FUNCTION_BLOCK RemoveAllMoverFromGroup EXTENDS TaskBase
VAR_INPUT
END_VAR
VAR_OUTPUT
END_VAR
VAR
	RemoveAllFromGrp			: MC_UngroupAllAxes;
	_caGroup			: ICollisionGroup;
	_removeAllMovers : BOOL;
	_errorId: UDINT;
	Logger : TcMessage_Ext;
END_VAR

METHOD Abort : BOOL
RemoveAllFromGrp.Execute := FALSE;
Abort := true;
State := 0;
END_METHOD

METHOD Cycle : BOOL
VAR_INPUT
END_VAR
CASE State OF
	0:
		IF _removeAllMovers THEN
			_done := FALSE;
			_error := FALSE;
			_busy := TRUE;
			RemoveAllFromGrp.Execute := TRUE;
			IF RemoveAllFromGrp.Busy THEN
				_removeAllMovers := FALSE;
				State := 10;
				logger.Send(TC_EVENTS.XtsCAGroupEvents.CAGroupRemoving,'');
			END_IF
		END_IF
		
	10:
		IF NOT RemoveAllFromGrp.Busy THEN
			IF RemoveAllFromGrp.Done THEN
				_done := TRUE;
				logger.Send(TC_EVENTS.XtsCAGroupEvents.AllMoversRemoved,'');
			ELSIF RemoveAllFromGrp.Error THEN
				_error := TRUE;
				_errorId := RemoveAllFromGrp.ErrorId;
				Logger.Send(TC_EVENTS.XtsCAGroupEvents.CAGroupRemoveError,'');
			END_IF
			_busy := FALSE;
			RemoveAllFromGrp.Execute := false;
			State := 0;
		END_IF
END_CASE


RemoveAllFromGrp(AxesGroup := _caGroup.GroupRef);
END_METHOD

METHOD FB_init : BOOL
VAR_INPUT
	bInitRetains : BOOL; // if TRUE, the retain variables are initialized (warm start / cold start)
	bInCopyCode : BOOL;  // if TRUE, the instance afterwards gets moved into the copy code (online change)
	CAGroup : ICollisionGroup;	
END_VAR
_caGroup := CAGroup;
END_METHOD

METHOD RemoveAllMover : BOOL
RemoveAllMover := _removeAllMovers := true;
END_METHOD

END_FUNCTION_BLOCK

(* stored: Version 1.1.0.1, ProductVersion 3.1.4024.12
   POU RemoveAllMoverFromGroup: Id {1511d483-7397-4cd0-a6db-08dd652e8cbb}, SpecialFunc None
   Method Abort: Id {e7050a73-9e5f-49ae-8033-79483a14dcd8}
   Method Cycle: Id {c68e4170-0a2c-460f-9ca9-a0eca48c8c15}
   Method FB_init: Id {639b4db7-7f3c-417a-8c60-934c2a4c839a}
   Method RemoveAllMover: Id {0b41790b-140c-4897-91fc-096c85c5f45b} *)
